(* Logix 5000 project; controller LeakTestAuto vendor 1 type 14 code 226 rev 37.11; software revision 37.01; part 8 of 13 *)
(* tags used below, declared in another part *)
   AOI_Barcode_Comms : AOI_CommStatus;
   AOI_CTS1 : AOI_CTS_INSTRUMENT;
   AOI_CTS1_Comms : AOI_CommStatus;
   AOI_CTS1_Seq : AOI_Sequencer_x64;
   AOI_CTS2 : AOI_CTS_INSTRUMENT;
   AOI_CTS2_Comms : AOI_CommStatus;
   AOI_CTS2_Seq : AOI_Sequencer_x64;
   AOI_Robot_Comms : AOI_CommStatus;
   AOI_SeqSteps : AOI_StandardSeqSteps;
   AOI_SRX100 : AOI_KeyenceBarcode;
   Barcode_ResultData : STR_Barcode;
   BarcodeInputs : udt_KeyenceScannerInputs;
   BarcodeOutputs : udt_KeyenceScannerOutputs;
   BarcodeScanner : udt_OutputStructure;
   CTS1_BarcodeWrite : STRING80;
   CTS1_BasicResult : MESSAGE;
   CTS1_DataRead : STRING80;
   CTS1_DetailResult : MESSAGE;
   CTS1_Inputs : udt_CTS_INPUTS_FROM;
   CTS1_LastResultEval : STRING16;
   CTS1_LastTestUID : DINT;
   CTS1_NextTestUID : DINT;
   CTS1_NumTestsInSeq : SINT;
   CTS1_Outputs : udt_CTS_OUTPUTS_TO;
   CTS1_ReadMsg : MESSAGE;
   CTS1_Ready : DINT;
   CTS1_Result : udt_CTS_RESULT;
   CTS1_ResultHistoryLeak : udt_CTS_RESULT[10];
   CTS1_ResultHistoryVol : udt_CTS_RESULT[10];
   CTS1_Seq : udt_SequenceStructure_X64;
   CTS1_SeqUID : DINT;
   CTS1_UIDMsg : MESSAGE;
   CTS1_WriteMsg : MESSAGE;
   CTS2_BarcodeWrite : STRING80;
   CTS2_BasicResult : MESSAGE;
   CTS2_DataRead : STRING80;
   CTS2_DetailResult : MESSAGE;
   CTS2_Inputs : udt_CTS_INPUTS_FROM;
   CTS2_LastResultEval : STRING16;
   CTS2_LastTestUID : DINT;
   CTS2_NextTestUID : DINT;
   CTS2_NumTestsInSeq : SINT;
   CTS2_Outputs : udt_CTS_OUTPUTS_TO;
   CTS2_ReadMsg : MESSAGE;
   CTS2_Ready : DINT;
   CTS2_Result : udt_CTS_RESULT;
   CTS2_ResultHistoryLeak : udt_CTS_RESULT[10];
   CTS2_ResultHistoryVol : udt_CTS_RESULT[10];
   CTS2_Seq : udt_SequenceStructure_X64;
   CTS2_SeqUID : DINT;
   CTS2_UIDMsg : MESSAGE;
   CTS2_WriteMsg : MESSAGE;
   CTS_NoResult : udt_CTS_RESULT;
   CTS_ResultDump : udt_CTS_RESULT;
   CurrentDUTData : udt_DUTHistory[2];
   FFLU_CTS1Leak : CONTROL;
   FFLU_CTS1Vol : CONTROL;
   FFLU_CTS2Leak : CONTROL;
   FFLU_CTS2Vol : CONTROL;
   LeakTester1 : udt_OutputStructure;
   LeakTester2 : udt_OutputStructure;
   Mode_CapCTS : BOOL;
   Nest1Cylinder : udt_OutputStructure;
   Nest2Cylinder : udt_OutputStructure;
   ONS_CTS1ClearResultsBC : BOOL;
   ONS_CTS1GetResults : BOOL;
   ONS_CTS1ResultHistory : BOOL;
   ONS_CTS2ClearResultsBC : BOOL;
   ONS_CTS2GetResults : BOOL;
   ONS_CTS2ResultHistory : BOOL;
   OP220 : udt_Mode;
   RobotInputs : udt_EpsonInputs;
   TON_CTS1GetResultRetry : TIMER;
   TON_CTS1GetResultTimeout : TIMER;
   TON_CTS1NotGettingResultsTimeout : TIMER;
   TON_CTS1Trigger0 : TIMER;
   TON_CTS1Trigger1 : TIMER;
   TON_CTS1Trigger2 : TIMER;
   TON_CTS2GetResultRetry : TIMER;
   TON_CTS2GetResultTimeout : TIMER;
   TON_CTS2NotGettingResultsTimeout : TIMER;
   TON_CTS2Trigger0 : TIMER;
   TON_CTS2Trigger1 : TIMER;
   TON_CTS2Trigger2 : TIMER;
   I_OP220_N3_DUT_PRE_NEST_0 : ALIAS FOR Local:3:I.Pt00.Data;
   OP220_ConsumedFromMain : DINT[50];
   OP220_ConsumedFromMain_PurgeModeEn : BOOL;
   OP220_ConsumedFromMain_RobotPickupSafe : BOOL;
   OP220_ProducedForMain : DINT[50];
   PLC : AOI_PLC;
   Purge_Count_DN : BOOL;   // Purge Counter Completed
(* MainProgram, continued *)

ROUTINE R13_ProduceConsume   (* ladder *)
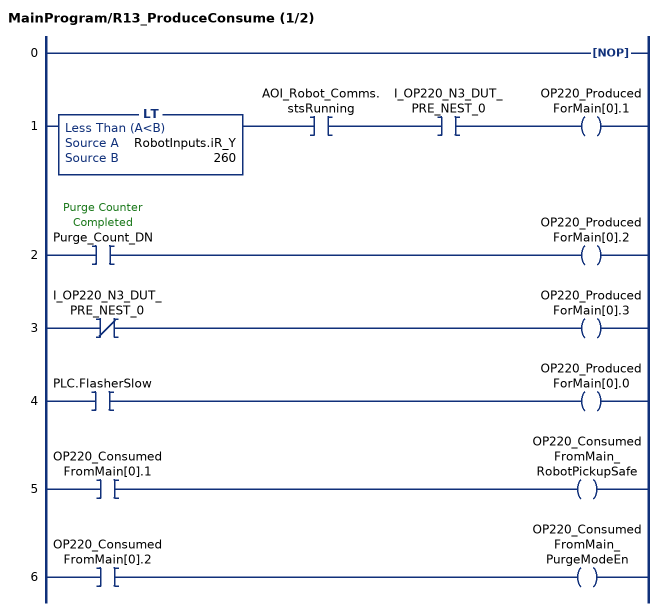
   0: NOP();
   1: LT(RobotInputs.iR_Y,260)XIC(AOI_Robot_Comms.stsRunning)XIC(I_OP220_N3_DUT_PRE_NEST_0)OTE(OP220_ProducedForMain[0].1);
   2: XIC(Purge_Count_DN)OTE(OP220_ProducedForMain[0].2);
   3: XIO(I_OP220_N3_DUT_PRE_NEST_0)OTE(OP220_ProducedForMain[0].3);
   4: XIC(PLC.FlasherSlow)OTE(OP220_ProducedForMain[0].0);
   5: XIC(OP220_ConsumedFromMain[0].1)OTE(OP220_ConsumedFromMain_RobotPickupSafe);
   6: XIC(OP220_ConsumedFromMain[0].2)OTE(OP220_ConsumedFromMain_PurgeModeEn);
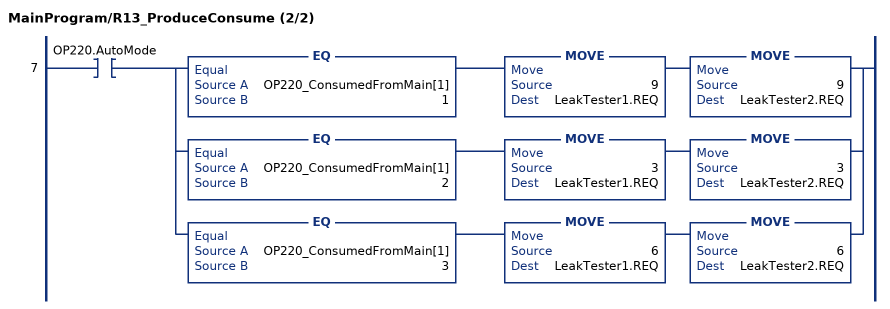
   7: XIC(OP220.AutoMode)[EQ(OP220_ConsumedFromMain[1],1) MOVE(9,LeakTester1.REQ) MOVE(9,LeakTester2.REQ) ,EQ(OP220_ConsumedFromMain[1],2) MOVE(3,LeakTester1.REQ) MOVE(3,LeakTester2.REQ) ,EQ(OP220_ConsumedFromMain[1],3) MOVE(6,LeakTester1.REQ) MOVE(6,LeakTester2.REQ) ];
END_ROUTINE

ROUTINE R20_Barcode   (* ladder *)
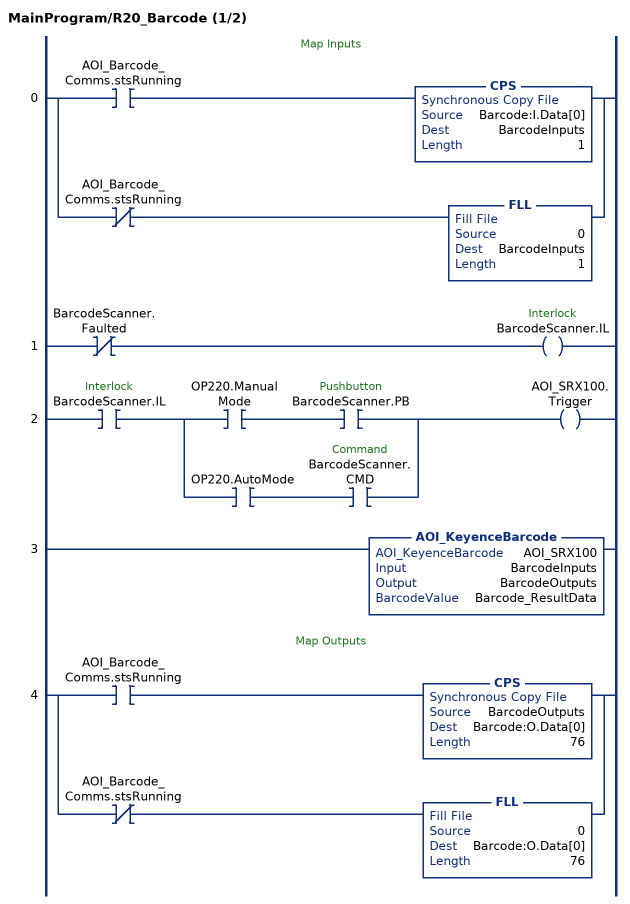
   // Map Inputs
   0: [XIC(AOI_Barcode_Comms.stsRunning) CPS(Barcode:I.Data[0],BarcodeInputs,1) ,XIO(AOI_Barcode_Comms.stsRunning) FLL(0,BarcodeInputs,1) ];
   1: XIO(BarcodeScanner.Faulted)OTE(BarcodeScanner.IL);
   2: XIC(BarcodeScanner.IL)[XIC(OP220.ManualMode) XIC(BarcodeScanner.PB) ,XIC(OP220.AutoMode) XIC(BarcodeScanner.CMD) ]OTE(AOI_SRX100.Trigger);
   3: AOI_KeyenceBarcode(AOI_SRX100,BarcodeInputs,BarcodeOutputs,Barcode_ResultData);
   // Map Outputs
   4: [XIC(AOI_Barcode_Comms.stsRunning) CPS(BarcodeOutputs,Barcode:O.Data[0],76) ,XIO(AOI_Barcode_Comms.stsRunning) FLL(0,Barcode:O.Data[0],76) ];
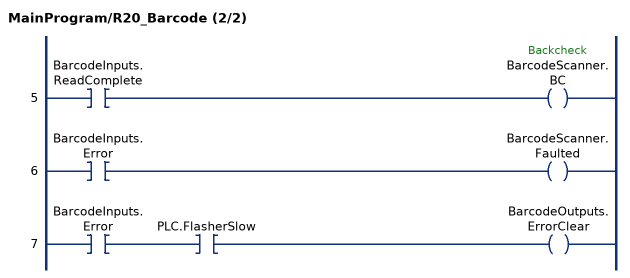
   5: XIC(BarcodeInputs.ReadComplete)OTE(BarcodeScanner.BC);
   6: XIC(BarcodeInputs.Error)OTE(BarcodeScanner.Faulted);
   7: XIC(BarcodeInputs.Error)XIC(PLC.FlasherSlow)OTE(BarcodeOutputs.ErrorClear);
END_ROUTINE

ROUTINE R30_LeakTester1   (* ladder *)
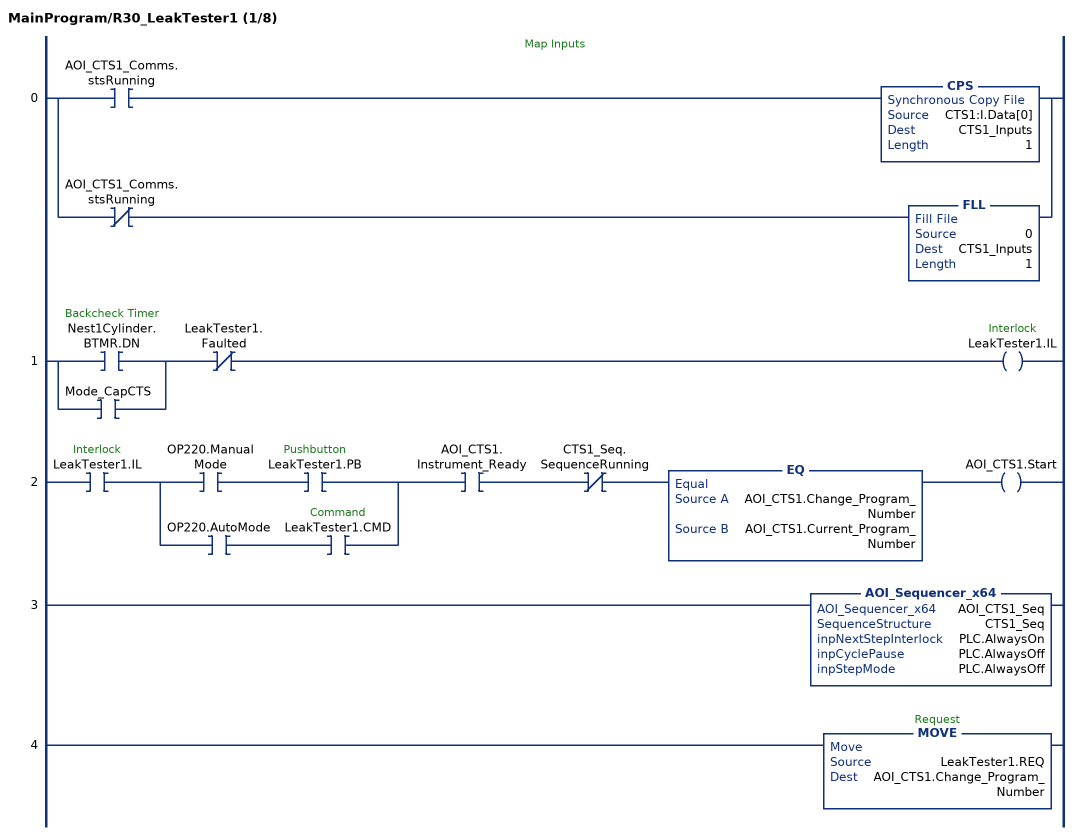
   // Map Inputs
   0: [XIC(AOI_CTS1_Comms.stsRunning) CPS(CTS1:I.Data[0],CTS1_Inputs,1) ,XIO(AOI_CTS1_Comms.stsRunning) FLL(0,CTS1_Inputs,1) ];
   1: [XIC(Nest1Cylinder.BTMR.DN) ,XIC(Mode_CapCTS) ]XIO(LeakTester1.Faulted)OTE(LeakTester1.IL);
   2: XIC(LeakTester1.IL)[XIC(OP220.ManualMode) XIC(LeakTester1.PB) ,XIC(OP220.AutoMode) XIC(LeakTester1.CMD) ]XIC(AOI_CTS1.Instrument_Ready)XIO(CTS1_Seq.SequenceRunning)EQ(AOI_CTS1.Change_Program_Number,AOI_CTS1.Current_Program_Number)OTE(AOI_CTS1.Start);
   3: AOI_Sequencer_x64(AOI_CTS1_Seq,CTS1_Seq,PLC.AlwaysOn,PLC.AlwaysOff,PLC.AlwaysOff);
   4: MOVE(LeakTester1.REQ,AOI_CTS1.Change_Program_Number);
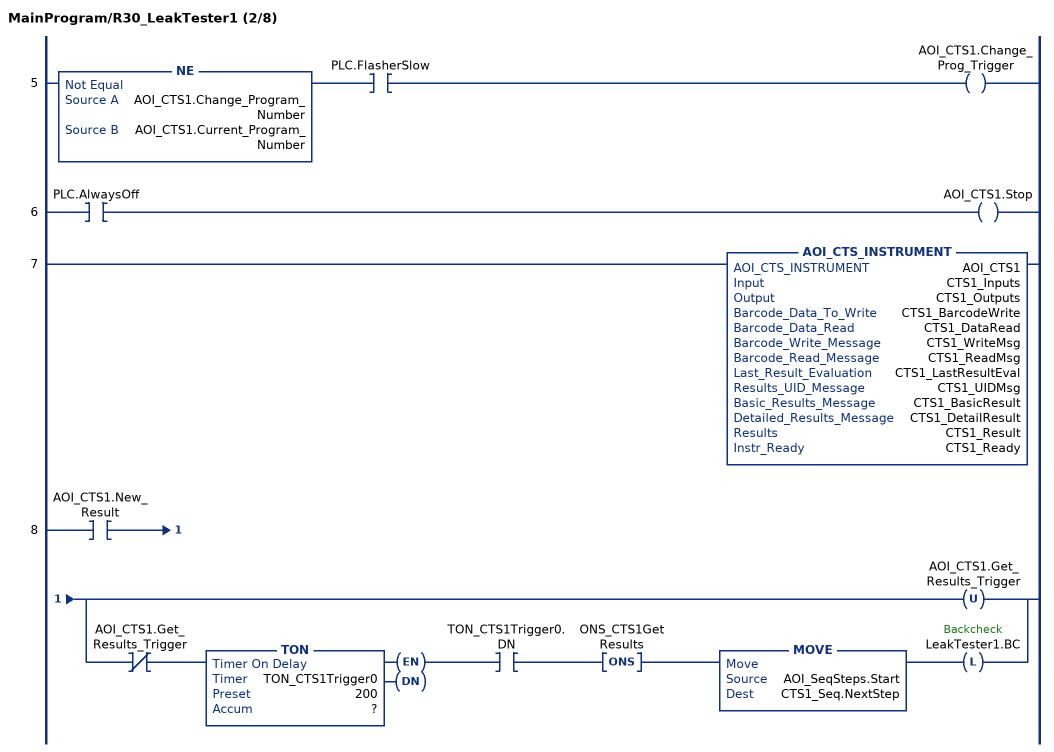
   5: NE(AOI_CTS1.Change_Program_Number,AOI_CTS1.Current_Program_Number)XIC(PLC.FlasherSlow)OTE(AOI_CTS1.Change_Prog_Trigger);
   6: XIC(PLC.AlwaysOff)OTE(AOI_CTS1.Stop);
   7: AOI_CTS_INSTRUMENT(AOI_CTS1,CTS1_Inputs,CTS1_Outputs,CTS1_BarcodeWrite,CTS1_DataRead,CTS1_WriteMsg,CTS1_ReadMsg,CTS1_LastResultEval,CTS1_UIDMsg,CTS1_BasicResult,CTS1_DetailResult,CTS1_Result,CTS1_Ready);
   8: XIC(AOI_CTS1.New_Result)[OTU(AOI_CTS1.Get_Results_Trigger) ,XIO(AOI_CTS1.Get_Results_Trigger) TON(TON_CTS1Trigger0,?,?) XIC(TON_CTS1Trigger0.DN) ONS(ONS_CTS1GetResults) MOVE(AOI_SeqSteps.Start,CTS1_Seq.NextStep) OTL(LeakTester1.BC) ];
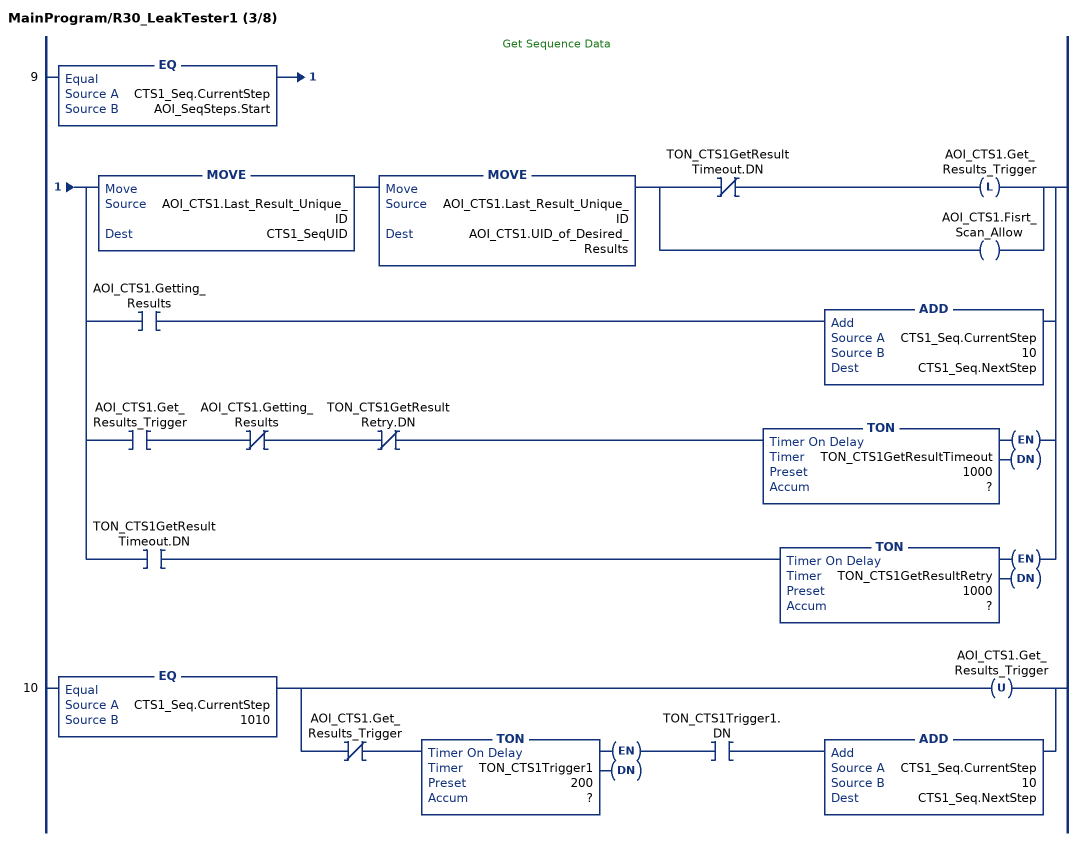
   // Get Sequence Data
   9: EQ(CTS1_Seq.CurrentStep,AOI_SeqSteps.Start)[MOVE(AOI_CTS1.Last_Result_Unique_ID,CTS1_SeqUID) MOVE(AOI_CTS1.Last_Result_Unique_ID,AOI_CTS1.UID_of_Desired_Results) [XIO(TON_CTS1GetResultTimeout.DN) OTL(AOI_CTS1.Get_Results_Trigger) ,OTE(AOI_CTS1.Fisrt_Scan_Allow) ] ,XIC(AOI_CTS1.Getting_Results) ADD(CTS1_Seq.CurrentStep,10,CTS1_Seq.NextStep) ,XIC(AOI_CTS1.Get_Results_Trigger) XIO(AOI_CTS1.Getting_Results) XIO(TON_CTS1GetResultRetry.DN) TON(TON_CTS1GetResultTimeout,?,?) ,XIC(TON_CTS1GetResultTimeout.DN) TON(TON_CTS1GetResultRetry,?,?) ];
   10: EQ(CTS1_Seq.CurrentStep,1010)[OTU(AOI_CTS1.Get_Results_Trigger) ,XIO(AOI_CTS1.Get_Results_Trigger) TON(TON_CTS1Trigger1,?,?) XIC(TON_CTS1Trigger1.DN) ADD(CTS1_Seq.CurrentStep,10,CTS1_Seq.NextStep) ];
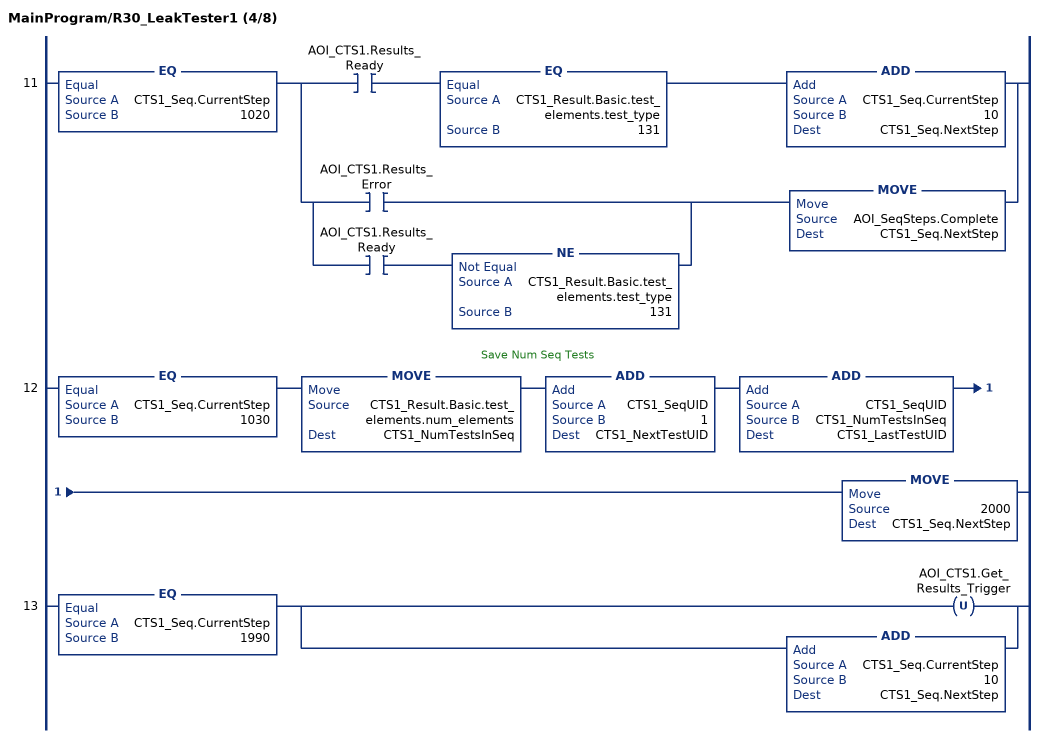
   11: EQ(CTS1_Seq.CurrentStep,1020)[XIC(AOI_CTS1.Results_Ready) EQ(CTS1_Result.Basic.test_elements.test_type,131) ADD(CTS1_Seq.CurrentStep,10,CTS1_Seq.NextStep) ,[XIC(AOI_CTS1.Results_Error) ,XIC(AOI_CTS1.Results_Ready) NE(CTS1_Result.Basic.test_elements.test_type,131) ] MOVE(AOI_SeqSteps.Complete,CTS1_Seq.NextStep) ];
   // Save Num Seq Tests
   12: EQ(CTS1_Seq.CurrentStep,1030)MOVE(CTS1_Result.Basic.test_elements.num_elements,CTS1_NumTestsInSeq)ADD(CTS1_SeqUID,1,CTS1_NextTestUID)ADD(CTS1_SeqUID,CTS1_NumTestsInSeq,CTS1_LastTestUID)MOVE(2000,CTS1_Seq.NextStep);
   13: EQ(CTS1_Seq.CurrentStep,1990)[OTU(AOI_CTS1.Get_Results_Trigger) ,ADD(CTS1_Seq.CurrentStep,10,CTS1_Seq.NextStep) ];
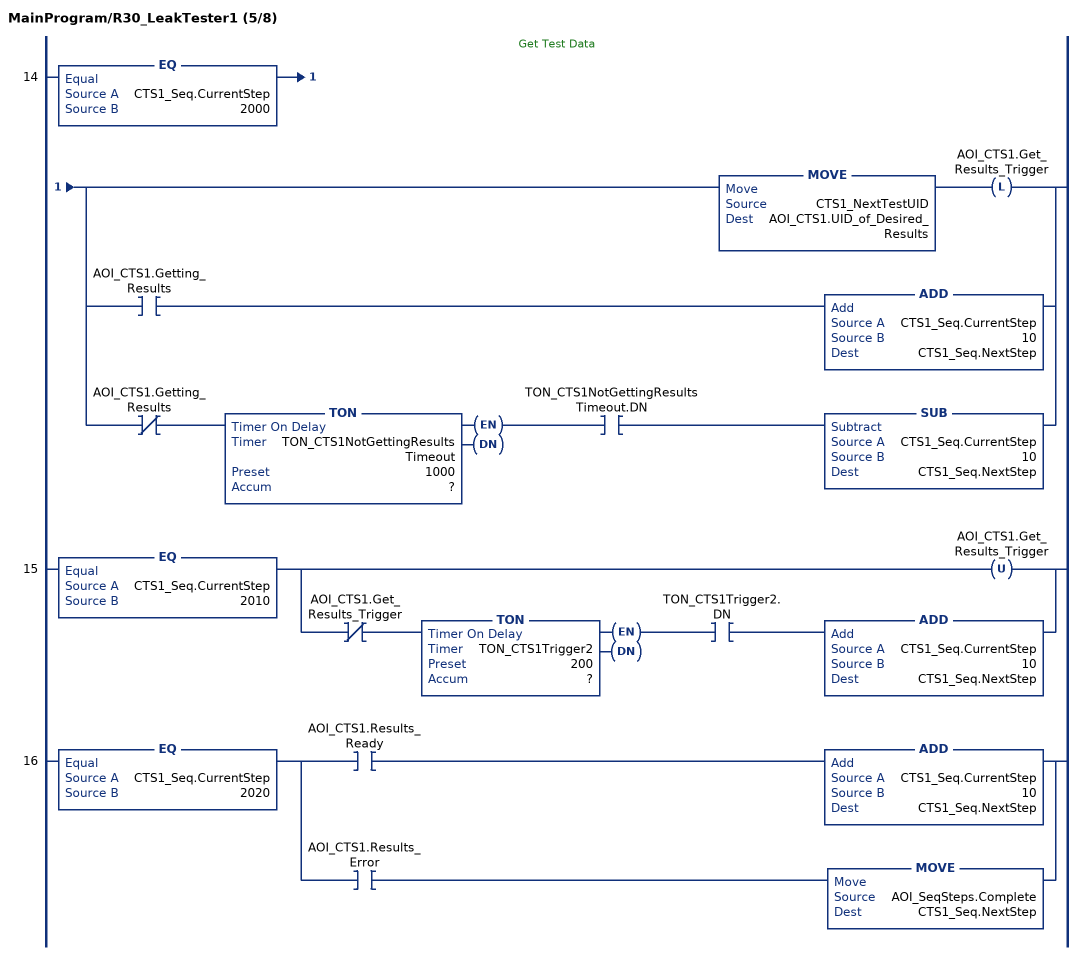
   // Get Test Data
   14: EQ(CTS1_Seq.CurrentStep,2000)[MOVE(CTS1_NextTestUID,AOI_CTS1.UID_of_Desired_Results) OTL(AOI_CTS1.Get_Results_Trigger) ,XIC(AOI_CTS1.Getting_Results) ADD(CTS1_Seq.CurrentStep,10,CTS1_Seq.NextStep) ,XIO(AOI_CTS1.Getting_Results) TON(TON_CTS1NotGettingResultsTimeout,?,?) XIC(TON_CTS1NotGettingResultsTimeout.DN) SUB(CTS1_Seq.CurrentStep,10,CTS1_Seq.NextStep) ];
   15: EQ(CTS1_Seq.CurrentStep,2010)[OTU(AOI_CTS1.Get_Results_Trigger) ,XIO(AOI_CTS1.Get_Results_Trigger) TON(TON_CTS1Trigger2,?,?) XIC(TON_CTS1Trigger2.DN) ADD(CTS1_Seq.CurrentStep,10,CTS1_Seq.NextStep) ];
   16: EQ(CTS1_Seq.CurrentStep,2020)[XIC(AOI_CTS1.Results_Ready) ADD(CTS1_Seq.CurrentStep,10,CTS1_Seq.NextStep) ,XIC(AOI_CTS1.Results_Error) MOVE(AOI_SeqSteps.Complete,CTS1_Seq.NextStep) ];
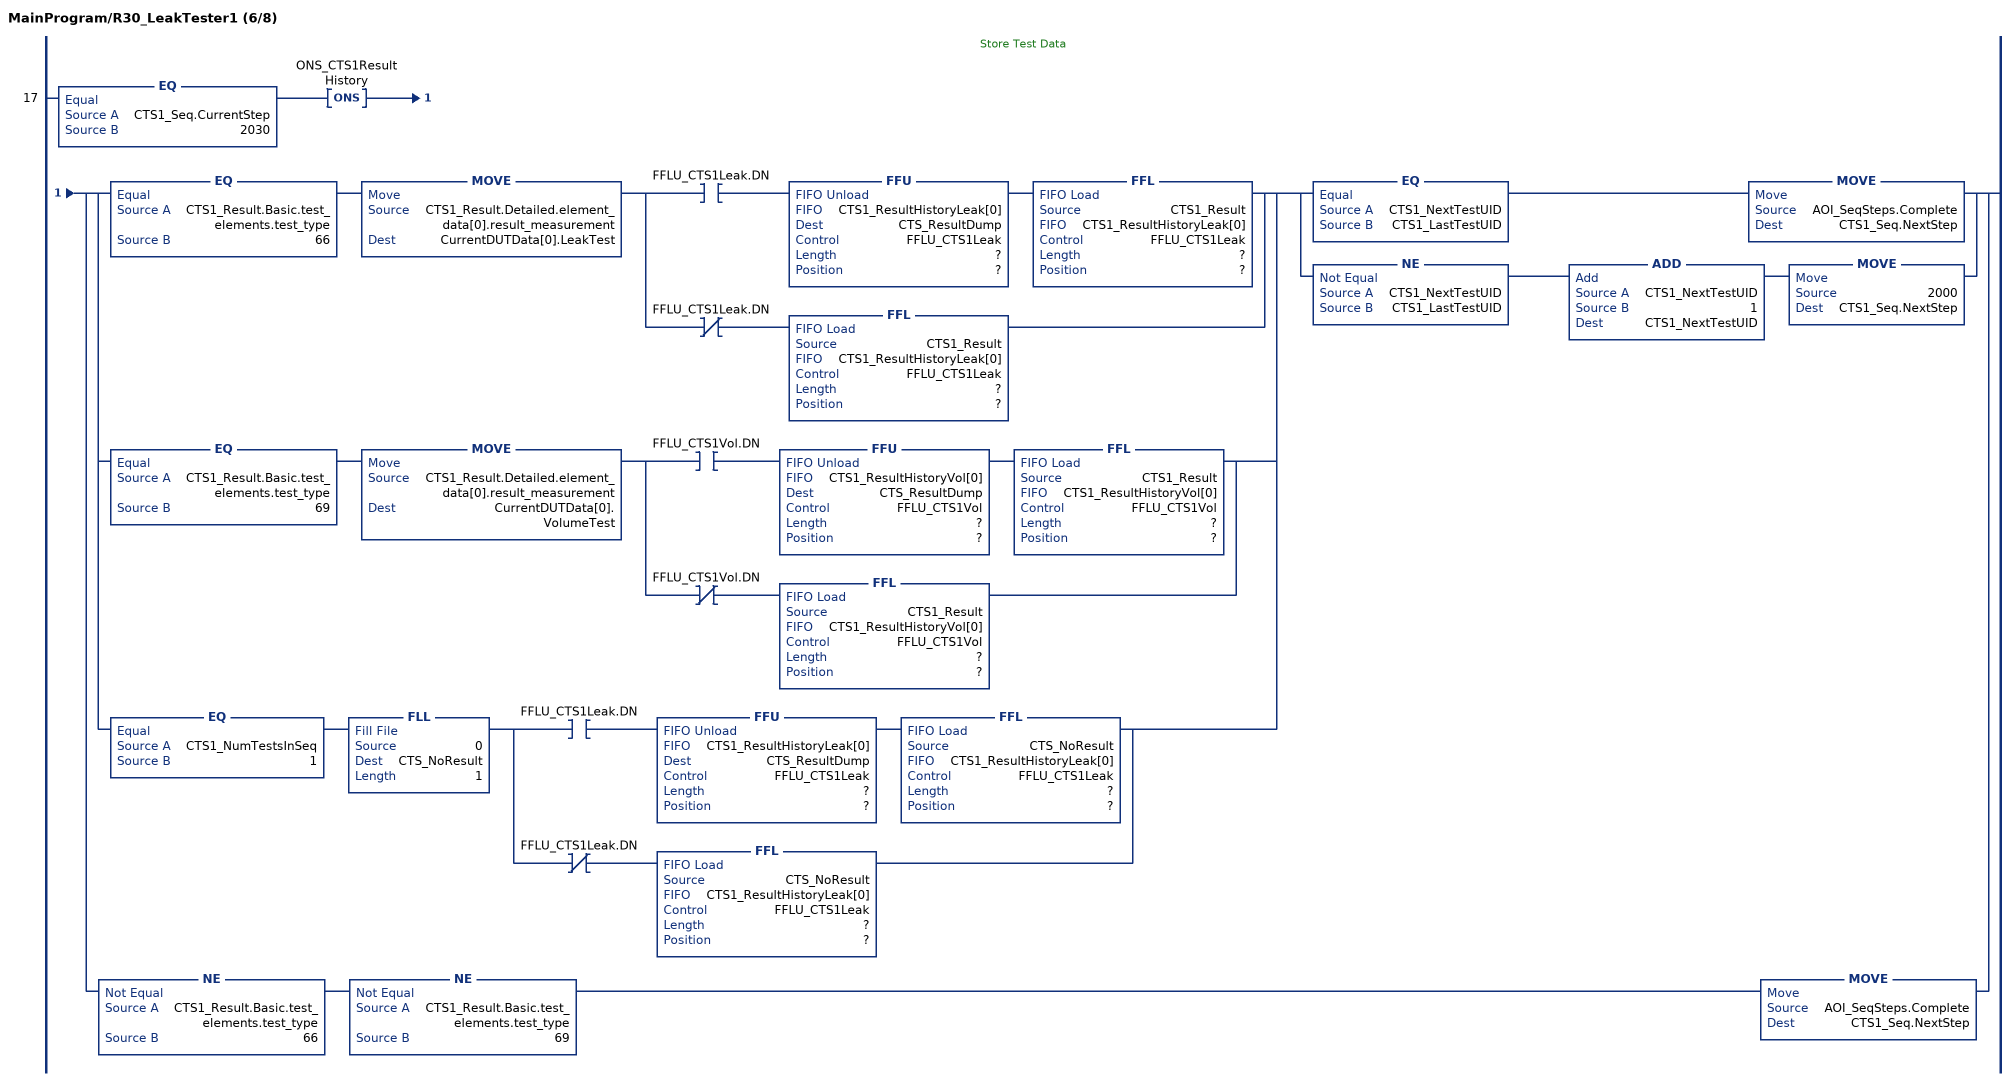
   // Store Test Data
   17: EQ(CTS1_Seq.CurrentStep,2030)ONS(ONS_CTS1ResultHistory)[[EQ(CTS1_Result.Basic.test_elements.test_type,66) MOVE(CTS1_Result.Detailed.element_data[0].result_measurement,CurrentDUTData[0].LeakTest) [XIC(FFLU_CTS1Leak.DN) FFU(CTS1_ResultHistoryLeak[0],CTS_ResultDump,FFLU_CTS1Leak,?,?) FFL(CTS1_Result,CTS1_ResultHistoryLeak[0],FFLU_CTS1Leak,?,?) ,XIO(FFLU_CTS1Leak.DN) FFL(CTS1_Result,CTS1_ResultHistoryLeak[0],FFLU_CTS1Leak,?,?) ] ,EQ(CTS1_Result.Basic.test_elements.test_type,69) MOVE(CTS1_Result.Detailed.element_data[0].result_measurement,CurrentDUTData[0].VolumeTest) [XIC(FFLU_CTS1Vol.DN) FFU(CTS1_ResultHistoryVol[0],CTS_ResultDump,FFLU_CTS1Vol,?,?) FFL(CTS1_Result,CTS1_ResultHistoryVol[0],FFLU_CTS1Vol,?,?) ,XIO(FFLU_CTS1Vol.DN) FFL(CTS1_Result,CTS1_ResultHistoryVol[0],FFLU_CTS1Vol,?,?) ] ,EQ(CTS1_NumTestsInSeq,1) FLL(0,CTS_NoResult,1) [XIC(FFLU_CTS1Leak.DN) FFU(CTS1_ResultHistoryLeak[0],CTS_ResultDump,FFLU_CTS1Leak,?,?) FFL(CTS_NoResult,CTS1_ResultHistoryLeak[0],FFLU_CTS1Leak,?,?) ,XIO(FFLU_CTS1Leak.DN) FFL(CTS_NoResult,CTS1_ResultHistoryLeak[0],FFLU_CTS1Leak,?,?) ] ] [EQ(CTS1_NextTestUID,CTS1_LastTestUID) MOVE(AOI_SeqSteps.Complete,CTS1_Seq.NextStep) ,NE(CTS1_NextTestUID,CTS1_LastTestUID) ADD(CTS1_NextTestUID,1,CTS1_NextTestUID) MOVE(2000,CTS1_Seq.NextStep) ] ,NE(CTS1_Result.Basic.test_elements.test_type,66) NE(CTS1_Result.Basic.test_elements.test_type,69) MOVE(AOI_SeqSteps.Complete,CTS1_Seq.NextStep) ];
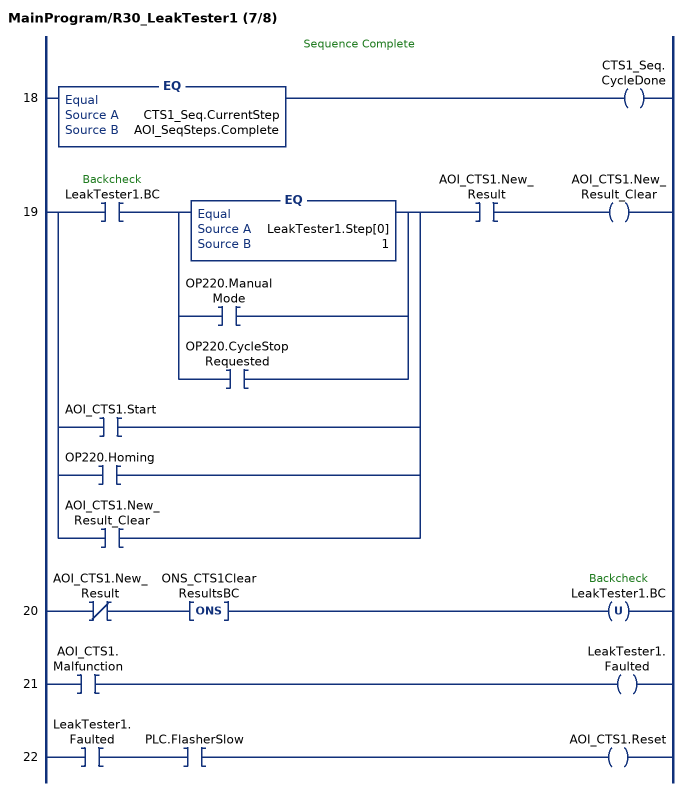
   // Sequence Complete
   18: EQ(CTS1_Seq.CurrentStep,AOI_SeqSteps.Complete)OTE(CTS1_Seq.CycleDone);
   19: [XIC(LeakTester1.BC) [EQ(LeakTester1.Step[0],1) ,XIC(OP220.ManualMode) ,XIC(OP220.CycleStopRequested) ] ,XIC(AOI_CTS1.Start) ,XIC(OP220.Homing) ,XIC(AOI_CTS1.New_Result_Clear) ]XIC(AOI_CTS1.New_Result)OTE(AOI_CTS1.New_Result_Clear);
   20: XIO(AOI_CTS1.New_Result)ONS(ONS_CTS1ClearResultsBC)OTU(LeakTester1.BC);
   21: XIC(AOI_CTS1.Malfunction)OTE(LeakTester1.Faulted);
   22: XIC(LeakTester1.Faulted)XIC(PLC.FlasherSlow)OTE(AOI_CTS1.Reset);
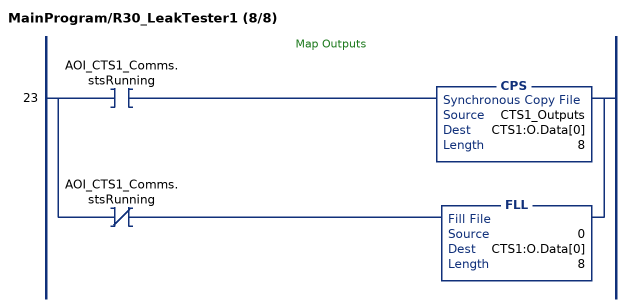
   // Map Outputs
   23: [XIC(AOI_CTS1_Comms.stsRunning) CPS(CTS1_Outputs,CTS1:O.Data[0],8) ,XIO(AOI_CTS1_Comms.stsRunning) FLL(0,CTS1:O.Data[0],8) ];
END_ROUTINE

ROUTINE R31_LeakTester2   (* ladder *)
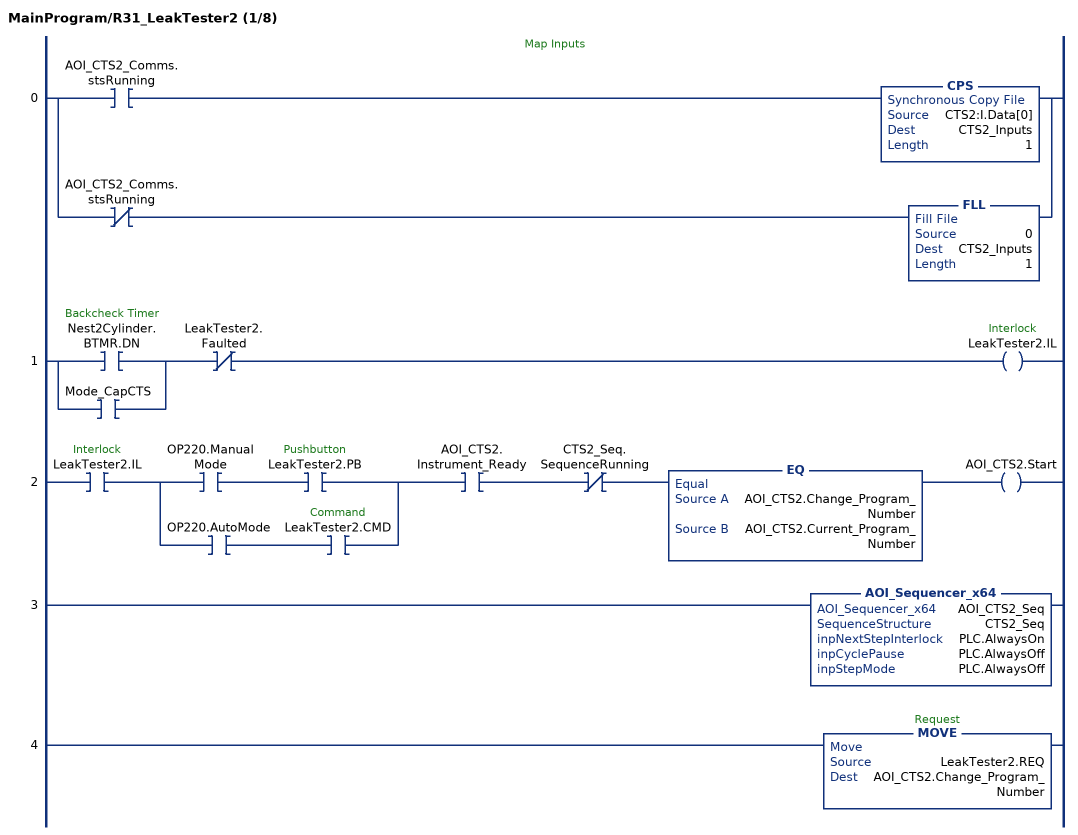
   // Map Inputs
   0: [XIC(AOI_CTS2_Comms.stsRunning) CPS(CTS2:I.Data[0],CTS2_Inputs,1) ,XIO(AOI_CTS2_Comms.stsRunning) FLL(0,CTS2_Inputs,1) ];
   1: [XIC(Nest2Cylinder.BTMR.DN) ,XIC(Mode_CapCTS) ]XIO(LeakTester2.Faulted)OTE(LeakTester2.IL);
   2: XIC(LeakTester2.IL)[XIC(OP220.ManualMode) XIC(LeakTester2.PB) ,XIC(OP220.AutoMode) XIC(LeakTester2.CMD) ]XIC(AOI_CTS2.Instrument_Ready)XIO(CTS2_Seq.SequenceRunning)EQ(AOI_CTS2.Change_Program_Number,AOI_CTS2.Current_Program_Number)OTE(AOI_CTS2.Start);
   3: AOI_Sequencer_x64(AOI_CTS2_Seq,CTS2_Seq,PLC.AlwaysOn,PLC.AlwaysOff,PLC.AlwaysOff);
   4: MOVE(LeakTester2.REQ,AOI_CTS2.Change_Program_Number);
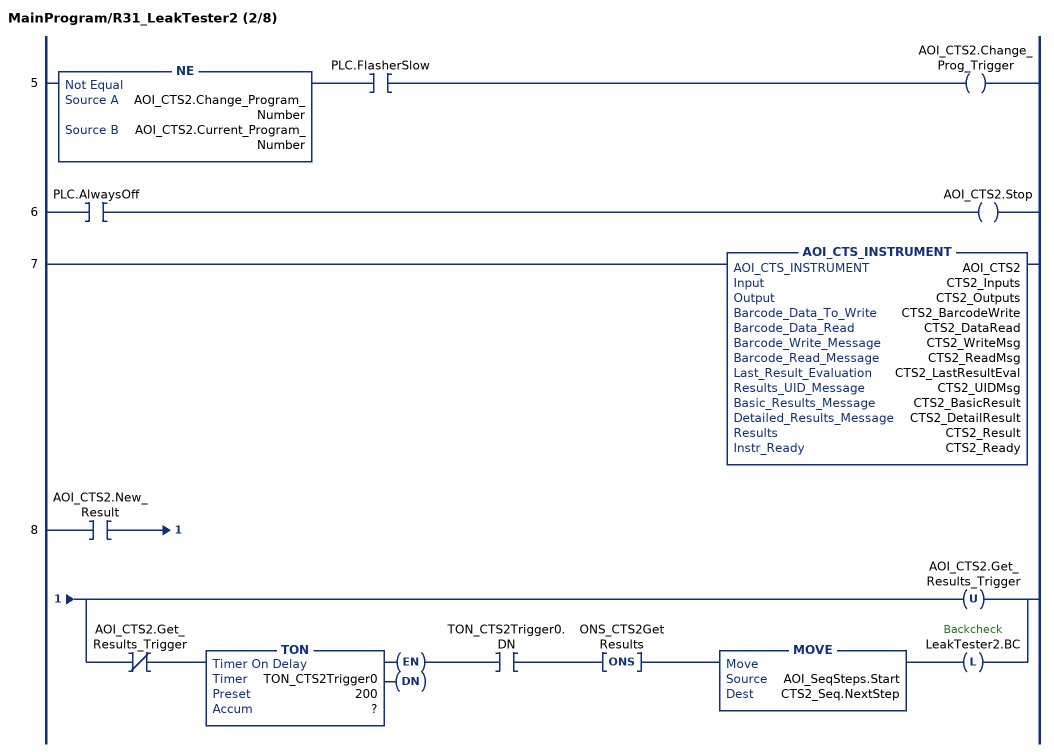
   5: NE(AOI_CTS2.Change_Program_Number,AOI_CTS2.Current_Program_Number)XIC(PLC.FlasherSlow)OTE(AOI_CTS2.Change_Prog_Trigger);
   6: XIC(PLC.AlwaysOff)OTE(AOI_CTS2.Stop);
   7: AOI_CTS_INSTRUMENT(AOI_CTS2,CTS2_Inputs,CTS2_Outputs,CTS2_BarcodeWrite,CTS2_DataRead,CTS2_WriteMsg,CTS2_ReadMsg,CTS2_LastResultEval,CTS2_UIDMsg,CTS2_BasicResult,CTS2_DetailResult,CTS2_Result,CTS2_Ready);
   8: XIC(AOI_CTS2.New_Result)[OTU(AOI_CTS2.Get_Results_Trigger) ,XIO(AOI_CTS2.Get_Results_Trigger) TON(TON_CTS2Trigger0,?,?) XIC(TON_CTS2Trigger0.DN) ONS(ONS_CTS2GetResults) MOVE(AOI_SeqSteps.Start,CTS2_Seq.NextStep) OTL(LeakTester2.BC) ];
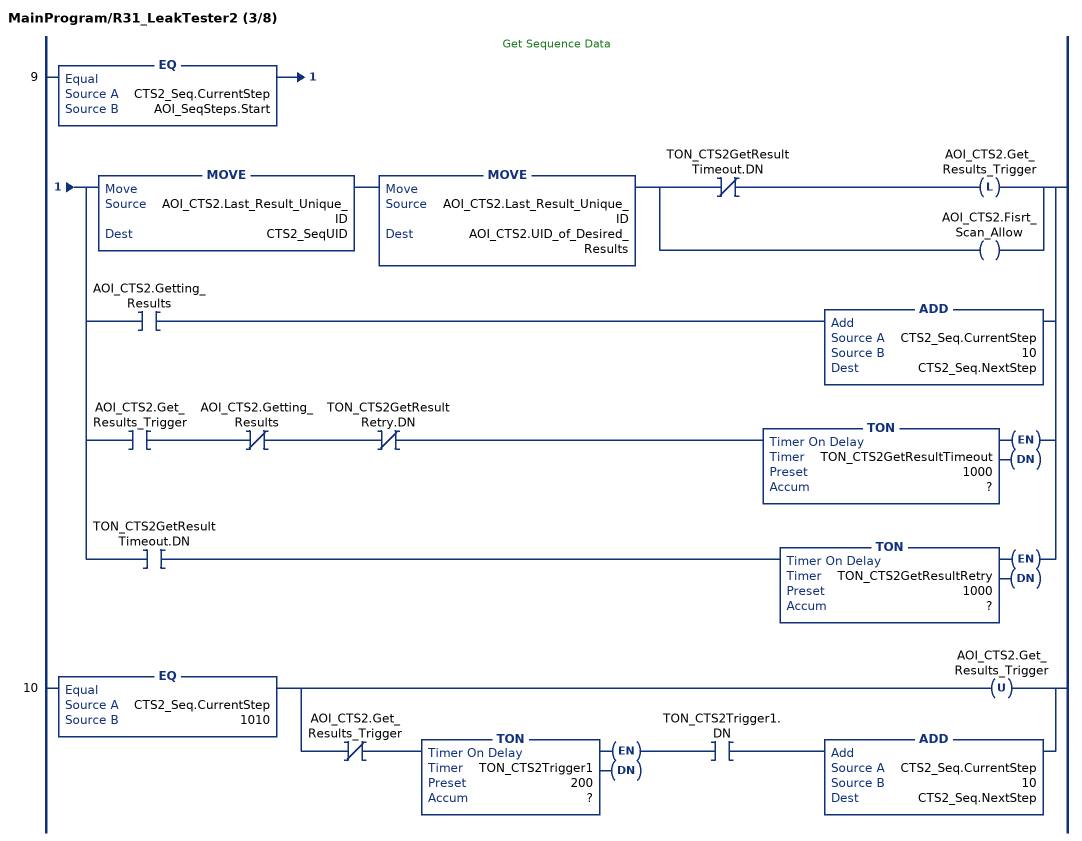
   // Get Sequence Data
   9: EQ(CTS2_Seq.CurrentStep,AOI_SeqSteps.Start)[MOVE(AOI_CTS2.Last_Result_Unique_ID,CTS2_SeqUID) MOVE(AOI_CTS2.Last_Result_Unique_ID,AOI_CTS2.UID_of_Desired_Results) [XIO(TON_CTS2GetResultTimeout.DN) OTL(AOI_CTS2.Get_Results_Trigger) ,OTE(AOI_CTS2.Fisrt_Scan_Allow) ] ,XIC(AOI_CTS2.Getting_Results) ADD(CTS2_Seq.CurrentStep,10,CTS2_Seq.NextStep) ,XIC(AOI_CTS2.Get_Results_Trigger) XIO(AOI_CTS2.Getting_Results) XIO(TON_CTS2GetResultRetry.DN) TON(TON_CTS2GetResultTimeout,?,?) ,XIC(TON_CTS2GetResultTimeout.DN) TON(TON_CTS2GetResultRetry,?,?) ];
   10: EQ(CTS2_Seq.CurrentStep,1010)[OTU(AOI_CTS2.Get_Results_Trigger) ,XIO(AOI_CTS2.Get_Results_Trigger) TON(TON_CTS2Trigger1,?,?) XIC(TON_CTS2Trigger1.DN) ADD(CTS2_Seq.CurrentStep,10,CTS2_Seq.NextStep) ];
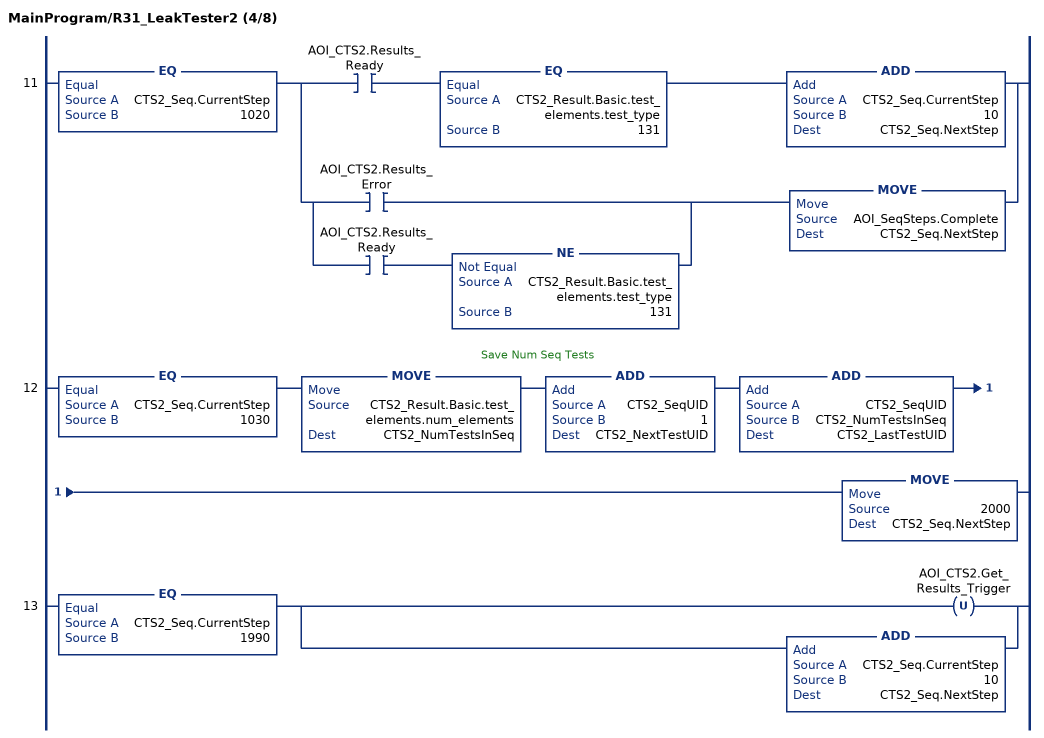
   11: EQ(CTS2_Seq.CurrentStep,1020)[XIC(AOI_CTS2.Results_Ready) EQ(CTS2_Result.Basic.test_elements.test_type,131) ADD(CTS2_Seq.CurrentStep,10,CTS2_Seq.NextStep) ,[XIC(AOI_CTS2.Results_Error) ,XIC(AOI_CTS2.Results_Ready) NE(CTS2_Result.Basic.test_elements.test_type,131) ] MOVE(AOI_SeqSteps.Complete,CTS2_Seq.NextStep) ];
   // Save Num Seq Tests
   12: EQ(CTS2_Seq.CurrentStep,1030)MOVE(CTS2_Result.Basic.test_elements.num_elements,CTS2_NumTestsInSeq)ADD(CTS2_SeqUID,1,CTS2_NextTestUID)ADD(CTS2_SeqUID,CTS2_NumTestsInSeq,CTS2_LastTestUID)MOVE(2000,CTS2_Seq.NextStep);
   13: EQ(CTS2_Seq.CurrentStep,1990)[OTU(AOI_CTS2.Get_Results_Trigger) ,ADD(CTS2_Seq.CurrentStep,10,CTS2_Seq.NextStep) ];
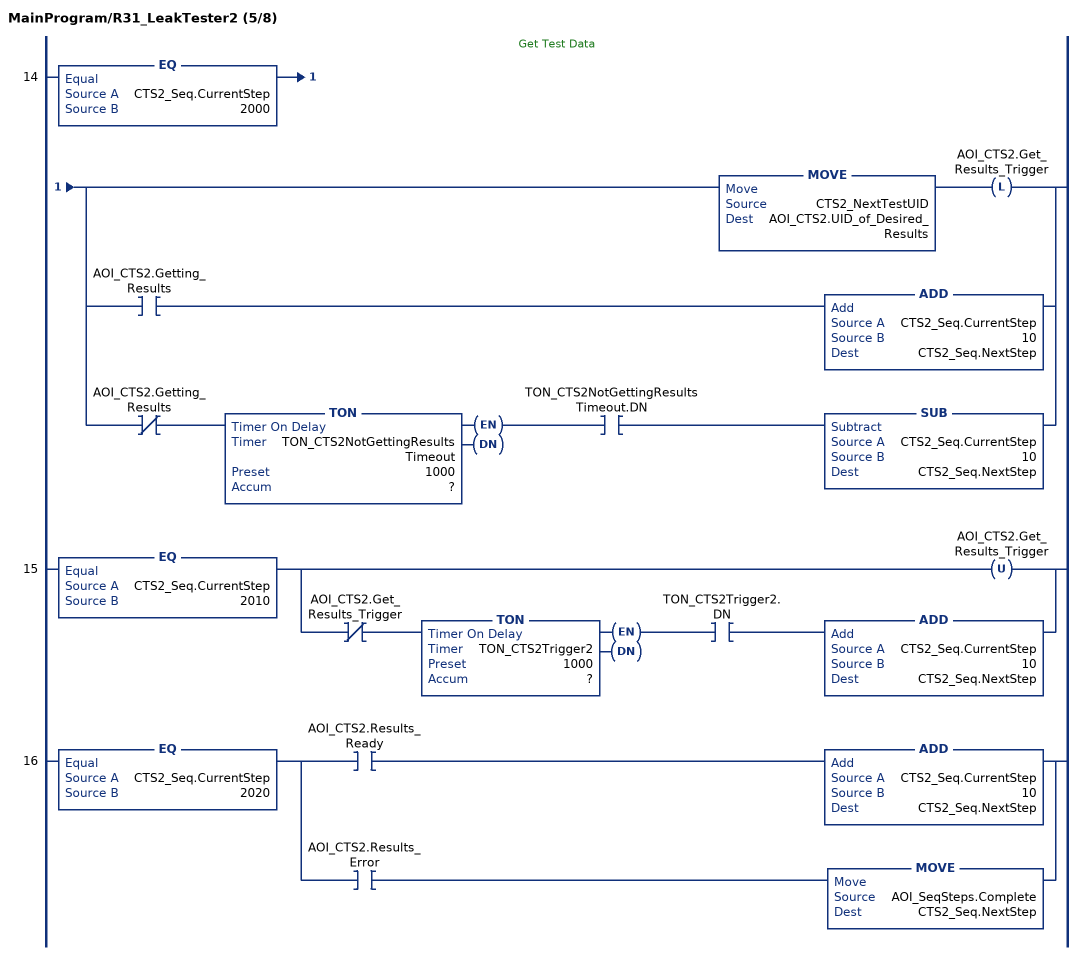
   // Get Test Data
   14: EQ(CTS2_Seq.CurrentStep,2000)[MOVE(CTS2_NextTestUID,AOI_CTS2.UID_of_Desired_Results) OTL(AOI_CTS2.Get_Results_Trigger) ,XIC(AOI_CTS2.Getting_Results) ADD(CTS2_Seq.CurrentStep,10,CTS2_Seq.NextStep) ,XIO(AOI_CTS2.Getting_Results) TON(TON_CTS2NotGettingResultsTimeout,?,?) XIC(TON_CTS2NotGettingResultsTimeout.DN) SUB(CTS2_Seq.CurrentStep,10,CTS2_Seq.NextStep) ];
   15: EQ(CTS2_Seq.CurrentStep,2010)[OTU(AOI_CTS2.Get_Results_Trigger) ,XIO(AOI_CTS2.Get_Results_Trigger) TON(TON_CTS2Trigger2,?,?) XIC(TON_CTS2Trigger2.DN) ADD(CTS2_Seq.CurrentStep,10,CTS2_Seq.NextStep) ];
   16: EQ(CTS2_Seq.CurrentStep,2020)[XIC(AOI_CTS2.Results_Ready) ADD(CTS2_Seq.CurrentStep,10,CTS2_Seq.NextStep) ,XIC(AOI_CTS2.Results_Error) MOVE(AOI_SeqSteps.Complete,CTS2_Seq.NextStep) ];
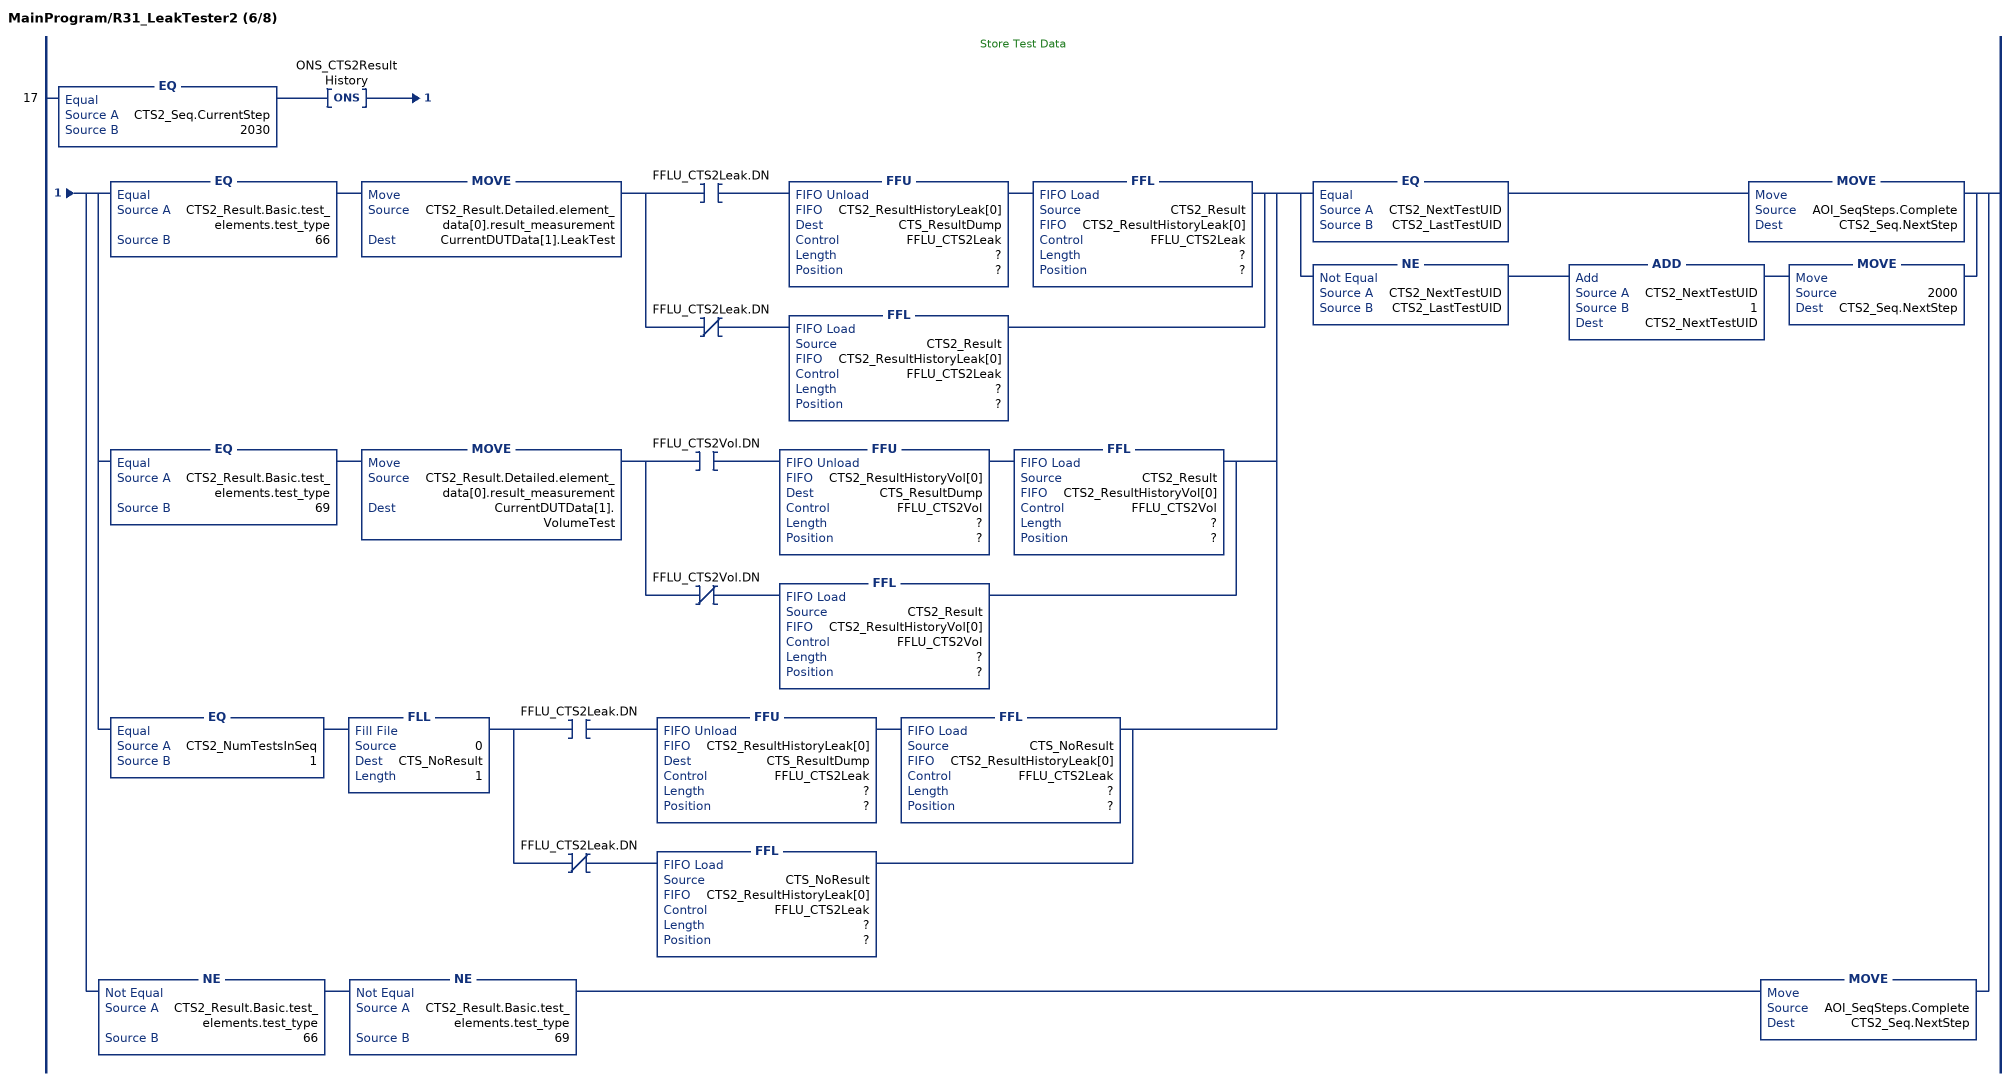
   // Store Test Data
   17: EQ(CTS2_Seq.CurrentStep,2030)ONS(ONS_CTS2ResultHistory)[[EQ(CTS2_Result.Basic.test_elements.test_type,66) MOVE(CTS2_Result.Detailed.element_data[0].result_measurement,CurrentDUTData[1].LeakTest) [XIC(FFLU_CTS2Leak.DN) FFU(CTS2_ResultHistoryLeak[0],CTS_ResultDump,FFLU_CTS2Leak,?,?) FFL(CTS2_Result,CTS2_ResultHistoryLeak[0],FFLU_CTS2Leak,?,?) ,XIO(FFLU_CTS2Leak.DN) FFL(CTS2_Result,CTS2_ResultHistoryLeak[0],FFLU_CTS2Leak,?,?) ] ,EQ(CTS2_Result.Basic.test_elements.test_type,69) MOVE(CTS2_Result.Detailed.element_data[0].result_measurement,CurrentDUTData[1].VolumeTest) [XIC(FFLU_CTS2Vol.DN) FFU(CTS2_ResultHistoryVol[0],CTS_ResultDump,FFLU_CTS2Vol,?,?) FFL(CTS2_Result,CTS2_ResultHistoryVol[0],FFLU_CTS2Vol,?,?) ,XIO(FFLU_CTS2Vol.DN) FFL(CTS2_Result,CTS2_ResultHistoryVol[0],FFLU_CTS2Vol,?,?) ] ,EQ(CTS2_NumTestsInSeq,1) FLL(0,CTS_NoResult,1) [XIC(FFLU_CTS2Leak.DN) FFU(CTS2_ResultHistoryLeak[0],CTS_ResultDump,FFLU_CTS2Leak,?,?) FFL(CTS_NoResult,CTS2_ResultHistoryLeak[0],FFLU_CTS2Leak,?,?) ,XIO(FFLU_CTS2Leak.DN) FFL(CTS_NoResult,CTS2_ResultHistoryLeak[0],FFLU_CTS2Leak,?,?) ] ] [EQ(CTS2_NextTestUID,CTS2_LastTestUID) MOVE(AOI_SeqSteps.Complete,CTS2_Seq.NextStep) ,NE(CTS2_NextTestUID,CTS2_LastTestUID) ADD(CTS2_NextTestUID,1,CTS2_NextTestUID) MOVE(2000,CTS2_Seq.NextStep) ] ,NE(CTS2_Result.Basic.test_elements.test_type,66) NE(CTS2_Result.Basic.test_elements.test_type,69) MOVE(AOI_SeqSteps.Complete,CTS2_Seq.NextStep) ];
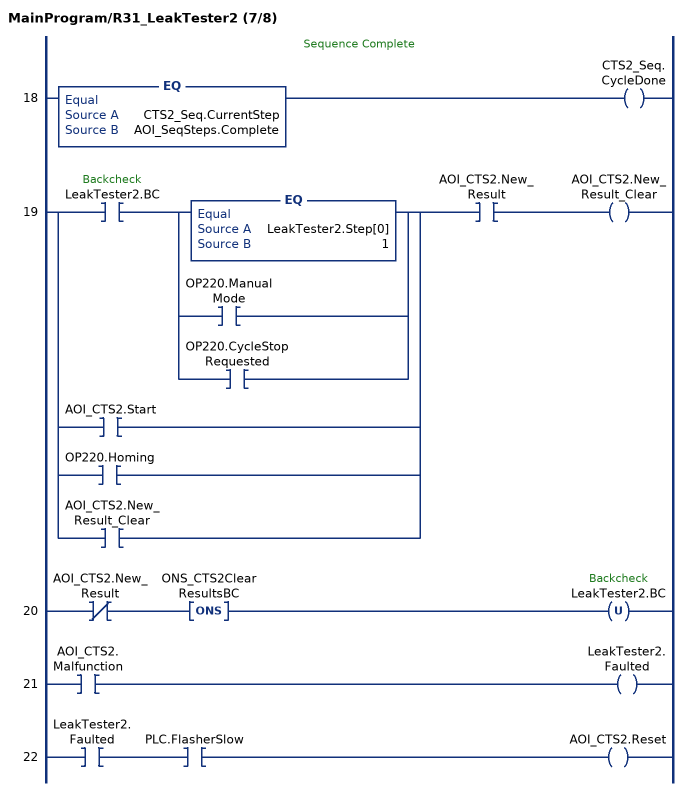
   // Sequence Complete
   18: EQ(CTS2_Seq.CurrentStep,AOI_SeqSteps.Complete)OTE(CTS2_Seq.CycleDone);
   19: [XIC(LeakTester2.BC) [EQ(LeakTester2.Step[0],1) ,XIC(OP220.ManualMode) ,XIC(OP220.CycleStopRequested) ] ,XIC(AOI_CTS2.Start) ,XIC(OP220.Homing) ,XIC(AOI_CTS2.New_Result_Clear) ]XIC(AOI_CTS2.New_Result)OTE(AOI_CTS2.New_Result_Clear);
   20: XIO(AOI_CTS2.New_Result)ONS(ONS_CTS2ClearResultsBC)OTU(LeakTester2.BC);
   21: XIC(AOI_CTS2.Malfunction)OTE(LeakTester2.Faulted);
   22: XIC(LeakTester2.Faulted)XIC(PLC.FlasherSlow)OTE(AOI_CTS2.Reset);
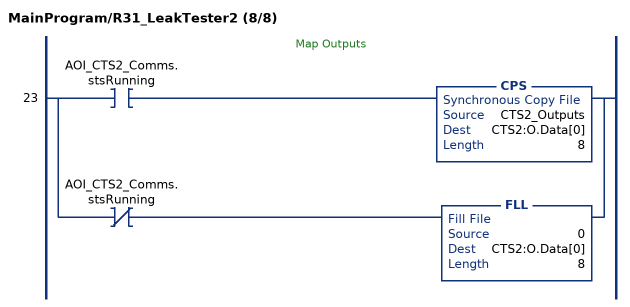
   // Map Outputs
   23: [XIC(AOI_CTS2_Comms.stsRunning) CPS(CTS2_Outputs,CTS2:O.Data[0],8) ,XIO(AOI_CTS2_Comms.stsRunning) FLL(0,CTS2:O.Data[0],8) ];
END_ROUTINE
